Fanuc KAREL source: kb00053.KL

-- PROVISIONAL review KL for V770-1; original PC SHA256 3627bfdc46e1c4d0b9fb8afd3f60078a1b7e67c9aa24dbbdbe6f65d79afc630f
-- Incomplete behavior may be omitted. Consult companion uncertainty JSON. Do not deploy.
PROGRAM KB00053
%NOLOCKGROUP
BEGIN
  -- UNRESOLVED_PC offsets 5-15; opcodes 27,31,75
  -- UNRESOLVED_PC offsets 20-24; opcodes 7F
END KB00053
